// TwinCAT 3 PLC project PLC851
// Title: UlyssesToolBox
// Company: HellWood
// ProjectVersion: 0.0.0.1
// ProgramVersion: 3.1.4024.0
// libraries:
//   CAA Memory, * (CAA Technical Workgroup)
//   Tc2_MC2, * (Beckhoff Automation GmbH)
//   Tc2_Standard, * (Beckhoff Automation GmbH)
//   Tc2_System, * (Beckhoff Automation GmbH)
//   Tc2_TcpIp, * (Beckhoff Automation GmbH)
//   Tc2_Utilities, * (Beckhoff Automation GmbH)
//   Tc3_DynamicMemory, * (Beckhoff Automation GmbH)
//   Tc3_MC2_AdvancedHoming, * (Beckhoff Automation GmbH)
//   Tc3_Module, * (Beckhoff Automation GmbH)
// project tree:
//   / MAIN.TcPOU, PlcTask.TcTTO
//   T04Connectivity/TCPIP/ FB_TcpSendReceive.TcPOU (not stored), FB_TcpSendReceiving.TcPOU (not stored), FB_TcpSendReceivingQueue.TcPOU (not stored)
//   T04Connectivity/TCPIP/SimpleClient/ SimpleTcpClient.TcPOU (not stored), stConnState.TcDUT, stSktPara.TcDUT (not stored)
//   T04Connectivity/TCPIP/TcpTaskQueue/ FB_SimpleTcpTaskQueue.TcPOU (not stored), ST_TcpTask.TcDUT (not stored), ST_TcpTaskBuffer.TcDUT (not stored)
//   T04Connectivity/TCPIP/TcpTaskQueue2/ FB_SimpleTcpTaskQueue2.TcPOU, ST_TcpTaskBuffer2.TcDUT, ST_TcpTask2.TcDUT
//   T05Motion/SimpleAxis/ E_MoveMode.TcDUT (not stored), E_SimpleAxisState.TcDUT (not stored), FB_SimpleAxis.TcPOU (not stored), ST_AxisSettings.TcDUT (not stored)
// real-time tasks:
//   TASK PlcTask: cycle T#10ms, priority 20, ADS port 350

CONFIGURATION PLC851
    RESOURCE PLC ON TwinCAT3
        TASK PlcTask(INTERVAL := T#10ms, PRIORITY := 20);
        PROGRAM MAIN WITH PlcTask : MAIN;
    END_RESOURCE
END_CONFIGURATION

// ---- T04Connectivity/TCPIP/SimpleClient/stConnState.TcDUT
TYPE stConnState :
STRUCT
	bConnected : BOOL;
	hSocket : T_HSOCKET;
	eState : E_SocketConnectionState;
	bError : BOOL;
	nErrId : UDINT;
END_STRUCT
END_TYPE

// ---- T04Connectivity/TCPIP/TcpTaskQueue2/ST_TcpTaskBuffer2.TcDUT
{attribute 'pack_mode' := '1'}
TYPE ST_TcpTaskBuffer2 :
STRUCT
	BufferInfo : UDINT;
	TaskData : ST_TcpTask2;
END_STRUCT
END_TYPE

// ---- T04Connectivity/TCPIP/TcpTaskQueue2/ST_TcpTask2.TcDUT
{attribute 'pack_mode' := '1'}
TYPE ST_TcpTask2 :
STRUCT
	TaskName : STRING(24);
	TaskType : INT; (* 0:Once, 1:Regular *)
	pData : PVOID;
	nData : UDINT;
END_STRUCT
END_TYPE

// ---- MAIN.TcPOU
PROGRAM MAIN
VAR
	tcpTest : FB_TcpSendReceivingQueue;
	tcpTest2 : FB_TcpSendReceiving;
	bAddTask: BOOL;
	arrData : ARRAY[0..255] OF BYTE;
	arrRecv : ARRAY[0..255] OF BYTE;
	bool1 : BOOL;
	bool2 : BOOL;
	dint1 : DINT;
	dint2 :DINT;
	STR1:STRING;
	MD5 : ARRAY[0..31] OF BYTE;
	MD5STR : STRING;
END_VAR

F_GenerateHashValue(
	hashMode:= Tc2_Utilities.E_HashMode.HASH_MD5, 
	pData:= ADR(STR1), 
	nData:= LEN(STR1), 
	pHash:= ADR(MD5), 
	nHash:= 16);

dint1 := 2030/100;
dint2 := 2030 MOD 100;
bool1 := FAILED(0);
bool2 := FAILED(16#80000013);
IF bAddTask THEN
	bAddTask := FALSE;
	arrData[0] := 67;
	tcpTest.AddTask('Send', 0, ADR(arrData), SIZEOF(arrData));
	tcpTest.AddTask('Send', 0, ADR(arrData), SIZEOF(arrData));
	tcpTest.AddTask('Send', 0, ADR(arrData), SIZEOF(arrData));
	tcpTest.AddTask('Send', 0, ADR(arrData), SIZEOF(arrData));
	tcpTest.AddTask('Send', 0, ADR(arrData), SIZEOF(arrData));
	arrData[0] := 68;
	tcpTest.AddTask('Send', 0, ADR(arrData), SIZEOF(arrData));
	tcpTest.AddTask('Send', 0, ADR(arrData), SIZEOF(arrData));
	tcpTest.AddTask('Send', 0, ADR(arrData), SIZEOF(arrData));
	tcpTest.AddTask('Send', 0, ADR(arrData), SIZEOF(arrData));
	tcpTest.AddTask('Send', 0, ADR(arrData), SIZEOF(arrData));
	arrData[0] := 69;
	tcpTest.AddTask('Send', 0, ADR(arrData), SIZEOF(arrData));
	tcpTest.AddTask('Send', 0, ADR(arrData), SIZEOF(arrData));
	tcpTest.AddTask('Send', 0, ADR(arrData), SIZEOF(arrData));
	tcpTest.AddTask('Send', 0, ADR(arrData), SIZEOF(arrData));
	tcpTest.AddTask('Send', 0, ADR(arrData), SIZEOF(arrData));
	arrData[0] := 70;
	tcpTest.AddTask('Send', 0, ADR(arrData), SIZEOF(arrData));
	tcpTest.AddTask('Send', 0, ADR(arrData), SIZEOF(arrData));
	tcpTest.AddTask('Send', 0, ADR(arrData), SIZEOF(arrData));
	tcpTest.AddTask('Send', 0, ADR(arrData), SIZEOF(arrData));
	tcpTest.AddTask('Send', 0, ADR(arrData), SIZEOF(arrData));
	arrData[0] := 71;
	tcpTest.AddTask('Send', 0, ADR(arrData), SIZEOF(arrData));
	tcpTest.AddTask('Send', 0, ADR(arrData), SIZEOF(arrData));
	tcpTest.AddTask('Send', 0, ADR(arrData), SIZEOF(arrData));
	tcpTest.AddTask('Send', 0, ADR(arrData), SIZEOF(arrData));
	tcpTest.AddTask('Send', 0, ADR(arrData), SIZEOF(arrData));
	arrData[0] := 72;
	tcpTest.AddTask('Send', 0, ADR(arrData), SIZEOF(arrData));
	tcpTest.AddTask('Send', 0, ADR(arrData), SIZEOF(arrData));
	tcpTest.AddTask('Send', 0, ADR(arrData), SIZEOF(arrData));
	tcpTest.AddTask('Send', 0, ADR(arrData), SIZEOF(arrData));
	tcpTest.AddTask('Send', 0, ADR(arrData), SIZEOF(arrData));
	arrData[0] := 73;
	tcpTest.AddTask('Send', 0, ADR(arrData), SIZEOF(arrData));
	tcpTest.AddTask('Send', 0, ADR(arrData), SIZEOF(arrData));
	tcpTest.AddTask('Send', 0, ADR(arrData), SIZEOF(arrData));
	tcpTest.AddTask('Send', 0, ADR(arrData), SIZEOF(arrData));
	tcpTest.AddTask('Send', 0, ADR(arrData), SIZEOF(arrData));
	arrData[0] := 74;
	tcpTest.AddTask('Send', 0, ADR(arrData), SIZEOF(arrData));
	tcpTest.AddTask('Send', 0, ADR(arrData), SIZEOF(arrData));
	tcpTest.AddTask('Send', 0, ADR(arrData), SIZEOF(arrData));
	tcpTest.AddTask('Send', 0, ADR(arrData), SIZEOF(arrData));
	tcpTest.AddTask('Send', 0, ADR(arrData), SIZEOF(arrData));
END_IF
tcpTest(
	bEnable:= TRUE, 
	bReset:= , 
	sRemoteIp:= '127.0.0.1', 
	nRemotePort:= 8003, 
	pRecvData:= ADR(arrRecv), 
	nRecvSize:= SIZEOF(arrRecv), 
	bBusyConnect=> , 
	bConnected=> , 
	bBusySend=> , 
	bSendDone=> , 
	bBusyRecv=> , 
	bRecvDone=> , 
	bError=> , 
	nRecvBytes=> , 
	bDataReceived=> );

END_PROGRAM

// ---- T04Connectivity/TCPIP/TcpTaskQueue2/FB_SimpleTcpTaskQueue2.TcPOU
FUNCTION_BLOCK FB_SimpleTcpTaskQueue2
VAR_INPUT
END_VAR
VAR_OUTPUT
END_VAR
VAR
	ActingQueue			: FB_MemRingBufferEx;
	ArrActingQueue		: ARRAY[0..MAXBUFFERSIZE] OF ST_TcpTaskBuffer2;
	
	fbMemMan			: FB_DynMem_Manager2;
	
	PushTask	: ST_TcpTask2;
	PopTask		: ST_TcpTask2;
	EmptyTask	: ST_TcpTask2;
	
	StepTaskConsume : DINT;
	
	_NoTaskToConsume : BOOL;
	_WaitingForTaskDone: BOOL;
	_ActingTaskCount: UDINT;
	_ActingUsedSize: UDINT;
	_ActingFreeSize: UDINT;
END_VAR
VAR CONSTANT
	MAXBUFFERSIZE: UDINT := 128;
END_VAR

_CyclicLogic();

METHOD PROTECTED _CyclicLogic : BOOL
VAR_INPUT
END_VAR
ActingQueue.A_GetFreeSize(pWrite:= , cbWrite:= , pBuffer:= ADR(ArrActingQueue), cbBuffer:= SIZEOF(ArrActingQueue), 
	bOk=> , pRead=> , cbRead=> , nCount=> _ActingTaskCount, cbSize=> _ActingUsedSize, cbFree=> _ActingFreeSize);
_NoTaskToConsume := (StepTaskConsume = 0);
_WaitingForTaskDone := (StepTaskConsume <> 0);
CASE StepTaskConsume OF
	0:
	_NoTaskToConsume := TRUE;
	IF ActingQueue.nCount <> 0 THEN
		StepTaskConsume := 10;
	END_IF
	
	10:
	ActingQueue.A_GetHead(pWrite:= , cbWrite:= , pBuffer:= ADR(ArrActingQueue), cbBuffer:= SIZEOF(ArrActingQueue), 
	bOk=> , pRead=> , cbRead=> , nCount=> _ActingTaskCount, cbSize=> _ActingUsedSize, cbFree=> _ActingFreeSize);
	IF ActingQueue.bOk THEN
		MEMCPY(destAddr:= ADR(PopTask), srcAddr:= ActingQueue.pRead, n:= MIN(SIZEOF(PopTask),ActingQueue.cbRead));
		StepTaskConsume := 20;
	ELSE
		StepTaskConsume := 0;
	END_IF
	
	20:
	// wait for task done
	
END_CASE
END_METHOD

PROPERTY ActingFreeSize : UDINT
GET
ActingFreeSize := _ActingFreeSize;
END_GET
END_PROPERTY

PROPERTY ActingTaskCount : UDINT
GET
ActingTaskCount := _ActingTaskCount;
END_GET
END_PROPERTY

PROPERTY ActingUsedSize : UDINT
GET
ActingUsedSize := _ActingUsedSize;
END_GET
END_PROPERTY

METHOD AddActingTask : BOOL
VAR_INPUT
	TaskName : STRING(24);
	TaskType : INT; (* 0:Once, 1:Regular *)
	pData : PVOID;
	nData : UDINT;
END_VAR
VAR
	pDynMem : PVOID;
END_VAR
IF nData > ActingQueue.cbFree THEN
	ADSLOGSTR(msgCtrlMask:= ADSLOG_MSGTYPE_ERROR OR ADSLOG_MSGTYPE_STRING , msgFmtStr:= 'AddTaskFailed: No free space', strArg:= '');
	RETURN;
END_IF
pDynMem := fbMemMan.Alloc(nSize:= nData, bReset:= TRUE);
MEMCPY(destAddr:= pDynMem, srcAddr:= pData, n:= nData);
PushTask.TaskName := TaskName;
PushTask.TaskType := TaskType;
PushTask.pData := pDynMem;
PushTask.nData := nData;
ActingQueue.A_AddTail(pWrite:= ADR(PushTask), cbWrite:= SIZEOF(PushTask), pBuffer:= ADR(ArrActingQueue), cbBuffer:= SIZEOF(ArrActingQueue), 
	bOk=> AddActingTask, pRead=> , cbRead=> , nCount=> _ActingTaskCount, cbSize=> _ActingUsedSize, cbFree=> _ActingFreeSize);
END_METHOD

PROPERTY CurrentTask : ST_TcpTask2
GET
CurrentTask := PopTask;
END_GET
END_PROPERTY

METHOD FinishTask : BOOL
VAR_INPUT
END_VAR
ActingQueue.A_FreeHead(pWrite:= , cbWrite:= , pBuffer:= ADR(ArrActingQueue), cbBuffer:= SIZEOF(ArrActingQueue), 
	bOk=> , pRead=> , cbRead=> , nCount=> _ActingTaskCount, cbSize=> _ActingUsedSize, cbFree=> _ActingFreeSize);
fbMemMan.Free2(PopTask.pData);
MEMCPY(destAddr:= ADR(PopTask), srcAddr:= ADR(EmptyTask), n:= SIZEOF(PopTask));
IF ActingQueue.bOk THEN
	IF ActingQueue.nCount <> 0 THEN
		StepTaskConsume := 10;
	ELSE
		StepTaskConsume := 0;
	END_IF
END_IF
END_METHOD

PROPERTY NoTaskToConsume : BOOL
GET
NoTaskToConsume := _NoTaskToConsume;
END_GET
END_PROPERTY

PROPERTY WaitingForTaskDone : BOOL
GET
WaitingForTaskDone := _WaitingForTaskDone;
END_GET
END_PROPERTY

END_FUNCTION_BLOCK
